(* PLC project Unnamed, Unknown Unnamed 1 *)
(* stored: creationDateTime 2019-08-06T14:23:42, modificationDateTime 2024-12-05T12:05:23 *)

PROGRAM MainStuff
  VAR
    csv_read_by_int0 : csv_read_by_int;
    CSV_ROWIDX : HMI_INT := 1;
    CSV_COLIDX : HMI_INT := 1;
    SAVE : HMI_BOOL := 0;
    CSV_ACK : HMI_BOOL;
    SEC_ACK : HMI_BOOL;
    CSV_RES : HMI_STRING;
    SEC_RES : HMI_STRING;
  END_VAR
  VAR_EXTERNAL
    FILENAME : HMI_STRING;
  END_VAR
  VAR
    CONTENT : HMI_STRING;
    csv_write_by_int0 : csv_write_by_int;
  END_VAR

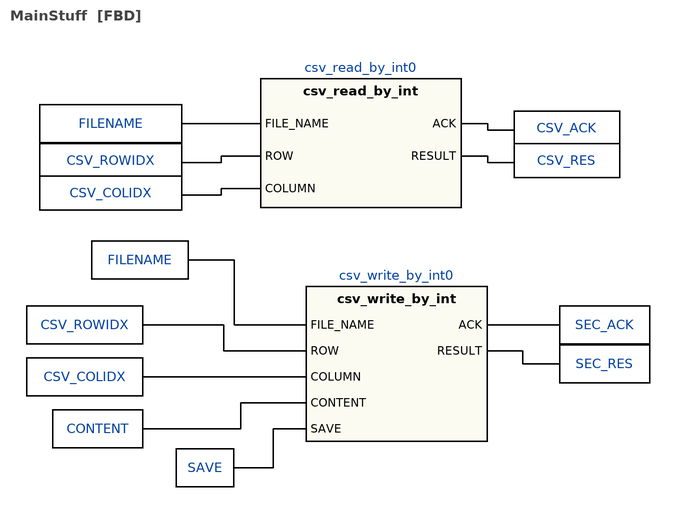
(* FBD diagram, written out as Structured Text *)
csv_read_by_int0(FILE_NAME := FILENAME, ROW := CSV_ROWIDX, COLUMN := CSV_COLIDX);
CSV_ACK := csv_read_by_int0.ACK;
CSV_RES := csv_read_by_int0.RESULT;
csv_write_by_int0(FILE_NAME := FILENAME, ROW := CSV_ROWIDX, COLUMN := CSV_COLIDX, CONTENT := CONTENT, SAVE := SAVE);
SEC_ACK := csv_write_by_int0.ACK;
SEC_RES := csv_write_by_int0.RESULT;
END_PROGRAM

CONFIGURATION config
  RESOURCE resource1 ON PLC
    TASK task0(INTERVAL := T#20ms, PRIORITY := 0);
    PROGRAM instance0 WITH task0 : MainStuff;
  END_RESOURCE
END_CONFIGURATION
